PROGRAM MAIN
VAR
	fbStarter		: FB_StarDeltaStarter;
END_VAR

fbStarter(
	bStart:= GVL.iStartPB, 
	bStop:= GVL.iStopPB, 
	tMainDelay:= T#1S, 
	tStarDeltaDelay:= T#5S, 
	bMainContactor=> GVL.oMainContactor, 
	bStarContactor=> GVL.oStarContactor, 
	bDeltaContactor=> GVL.oDeltaContactor,
	sStateDesciption => GVL.oState);

END_PROGRAM

(* stored: Version 1.1.0.1, ProductVersion 3.1.4024.10
   POU MAIN: Id {4d3cd65a-3d36-4163-b8ce-3aa108fddf81}, SpecialFunc None *)
